{attribute 'GeneratedUsingTerminal: EP1859-0042-0018'}
{attribute addProperty BoxType "EP1859-0042-0018"}
{attribute addProperty Id "EtcSlaveTerminalBaseDI_X01_Pin4AT %I*DI_X01_Pin_830843C11DI_X01_Pin2AT %I*DI_X01_Pin_830843C11DI_X02_Pin4AT %I*DI_X02_Pin_830843C11DI_X02_Pin2AT %I*DI_X02_Pin_830843C11DI_X03_Pin4AT %I*DI_X03_Pin_830843C11DI_X03_Pin2AT %I*DI_X03_Pin_830843C11DI_X04_Pin4AT %I*DI_X04_Pin_830843C11DI_X04_Pin2AT %I*DI_X04_Pin_830843C11DO_X05_Pin4AT %Q*DO_X05_Pin_42CA91F71DO_X05_Pin2AT %Q*DO_X05_Pin_42CA91F71DO_X06_Pin4AT %Q*DO_X06_Pin_42CA91F71DO_X06_Pin2AT %Q*DO_X06_Pin_42CA91F71DO_X07_Pin4AT %Q*DO_X07_Pin_42CA91F71DO_X07_Pin2AT %Q*DO_X07_Pin_42CA91F71DO_X08_Pin4AT %Q*DO_X08_Pin_42CA91F71DO_X08_Pin2AT %Q*DO_X08_Pin_42CA91F71WcStateAT %I*WcState_9091E0EB2InfoDataAT %I*InfoData_6F19DB2B2"}
{attribute addProperty CRC "2340578266"}
{attribute addProperty Size "20"}
TYPE EP1859_8B8263DA EXTENDS EtcSlaveTerminalBase :
STRUCT
	{attribute addProperty Name "DI_X01_Pin4"}
	DI_X01_Pin4 : DI_X01_Pin_830843C1;
	{attribute addProperty Name "DI_X01_Pin2"}
	DI_X01_Pin2 : DI_X01_Pin_830843C1;
	{attribute addProperty Name "DI_X02_Pin4"}
	DI_X02_Pin4 : DI_X02_Pin_830843C1;
	{attribute addProperty Name "DI_X02_Pin2"}
	DI_X02_Pin2 : DI_X02_Pin_830843C1;
	{attribute addProperty Name "DI_X03_Pin4"}
	DI_X03_Pin4 : DI_X03_Pin_830843C1;
	{attribute addProperty Name "DI_X03_Pin2"}
	DI_X03_Pin2 : DI_X03_Pin_830843C1;
	{attribute addProperty Name "DI_X04_Pin4"}
	DI_X04_Pin4 : DI_X04_Pin_830843C1;
	{attribute addProperty Name "DI_X04_Pin2"}
	DI_X04_Pin2 : DI_X04_Pin_830843C1;
	{attribute addProperty Name "DO_X05_Pin4"}
	DO_X05_Pin4 : DO_X05_Pin_42CA91F7;
	{attribute addProperty Name "DO_X05_Pin2"}
	DO_X05_Pin2 : DO_X05_Pin_42CA91F7;
	{attribute addProperty Name "DO_X06_Pin4"}
	DO_X06_Pin4 : DO_X06_Pin_42CA91F7;
	{attribute addProperty Name "DO_X06_Pin2"}
	DO_X06_Pin2 : DO_X06_Pin_42CA91F7;
	{attribute addProperty Name "DO_X07_Pin4"}
	DO_X07_Pin4 : DO_X07_Pin_42CA91F7;
	{attribute addProperty Name "DO_X07_Pin2"}
	DO_X07_Pin2 : DO_X07_Pin_42CA91F7;
	{attribute addProperty Name "DO_X08_Pin4"}
	DO_X08_Pin4 : DO_X08_Pin_42CA91F7;
	{attribute addProperty Name "DO_X08_Pin2"}
	DO_X08_Pin2 : DO_X08_Pin_42CA91F7;
	{attribute addProperty Name "WcState"}
	WcState : WcState_9091E0EB;
	{attribute addProperty Name "InfoData"}
	InfoData : InfoData_6F19DB2B;
END_STRUCT
END_TYPE

(* stored: Version 1.2.0.0, ProductVersion 3.1.4024.9
   DUT EP1859_8B8263DA: Id {9d3ac2df-b18e-4665-a408-3fb1c422b7e0} *)
